// TIA Portal V19 export
VAR_GLOBAL   // PLC tag table "Unit2"
END_VAR
VAR_GLOBAL CONSTANT   // user constants
   Unit2_NO_OF_EMs : Int := 6;   // 最高的Em号
   Unit2_EM0 : Int := 0;
   Unit2_EM1 : Int := 1;
   Unit2_EM2 : Int := 2;
   Unit2_EM3 : Int := 3;
   Unit2_EM4 : Int := 4;
   Unit2_EM5 : Int := 5;
   Unit2_EM6 : Int := 6;
END_VAR
